{attribute addProperty BoxType "KL9160"}
{attribute addProperty Id "Channel_1Channel_0970199100"}
{attribute addProperty CRC "2629167143"}
{attribute addProperty SizeInBites "0"}
{attribute addProperty SizeInBytes "0"}
TYPE KL9160_9CB5E827 :
STRUCT
	{attribute addProperty Name "Channel_1"}
	Channel_1 : Channel_09701991;
END_STRUCT
END_TYPE

(* stored: Version 1.2.0.0, ProductVersion 3.1.4024.9
   DUT KL9160_9CB5E827: Id {fa9c64a9-2bb3-4b7e-8b22-6749e400953d} *)
